// TIA Portal V20 export
TYPE "typeCmHmiInterface"
// stored: Access Published, Namespace Unit1.Em5
   STRUCT
      distance : "LER_typeDistanceInterface";
      softcam : "Unit1.Em5.typeCmHmiInterfaceSoftCam";
      brakeTest : "Unit1.Em5.typeCmHmiInterfaceBrakeTest";
   END_STRUCT;
   // distance.setValue.direction := TRUE;
   // distance.setValue.distancePTPSV := 4300.0;
END_TYPE
